FUNCTION_BLOCK Execute IMPLEMENTS ITF_PackMLState, ITF_States
VAR
	_MyContext : ITF_PackMLMachine;
	_MyNextState : ITF_PackMLState;
	_MyStoppingState : ITF_PackMLState;
	_MyAbortingState : ITF_PackMLState;
	_MyName : STRING(20) := 'Execute';
END_VAR

PROPERTY AbortingState : ITF_PackMLState
GET
AbortingState := _MyAbortingState;
END_GET
SET
_MyAbortingState := AbortingState;
END_SET
END_PROPERTY

METHOD CyclicLogic : BOOL
VAR_INPUT
END_VAR
END_METHOD

{warning 'add method implementation '}
METHOD EStop : BOOL
END_METHOD

{warning 'add property implementation'}
PROPERTY MyNextState : ITF_PackMLState
GET
MyNextState := _MyNextState;
END_GET
SET
_MyNextState := MyNextState;
END_SET
END_PROPERTY

PROPERTY MyStateName : String(20)
GET
MyStateName := _MyName;
END_GET
END_PROPERTY

{warning 'add method implementation '}
METHOD Reset : BOOL
END_METHOD

{warning 'add method implementation '}
METHOD SetContext : BOOL
VAR_INPUT
	context	: ITF_PackMLMachine;
END_VAR
_MyContext := context;
END_METHOD

{warning 'add method implementation '}
METHOD Start : BOOL
END_METHOD

{warning 'add method implementation '}
METHOD Stop : BOOL
END_METHOD

{warning 'add property implementation'}
PROPERTY StoppingState : ITF_PackMLState
GET
StoppingState := _MyStoppingState;
END_GET
SET
_MyStoppingState := StoppingState;
END_SET
END_PROPERTY

END_FUNCTION_BLOCK

(* stored: Version 1.1.0.1, ProductVersion 3.1.4024.12
   POU Execute: Id {16de238c-02d0-4654-b592-0c63039045d2}, SpecialFunc None
   Property AbortingState: Id {a5c15762-a08b-4161-91c2-5b5d8500ebc6}
   Get Get: Id {8849a4be-4f5c-408f-8893-220c57711478}
   Set Set: Id {d35cdb24-c26a-4df2-ac93-3d6a83189bfe}
   Method CyclicLogic: Id {ac050c99-a704-455e-9c5a-e556222f067a}
   Method EStop: Id {2ba6e0cd-1efe-4003-8123-65a9ba9b7ac2}
   Property MyNextState: Id {2d3d8db9-a44d-47ba-a9fd-8c0878cf2f5b}
   Get Get: Id {5d2e5776-26ac-4a8d-9a97-ef8b5054a217}
   Set Set: Id {b0111621-da13-46d4-85b1-9f62b318817a}
   Property MyStateName: Id {8976abae-eefc-4513-8348-4ffb6ed01903}
   Get Get: Id {0ffcb83e-153b-4248-94b8-c0ac0d69ac6e}
   Method Reset: Id {1a9cf0ec-8b14-4e8d-9539-992a9b7b2e78}
   Method SetContext: Id {1700c1be-96df-4ce8-8a27-f90db3bd76f2}
   Method Start: Id {42576e4a-c1d8-4012-9b36-1be3c4c250b5}
   Method Stop: Id {26dae254-0c3f-4d8e-8ed6-04c9be98f59b}
   Property StoppingState: Id {94f61d8a-f201-44ab-9c5d-1676d4b7878e}
   Get Get: Id {fcd83bcc-4566-4c4b-88c2-ce94446d7b5f}
   Set Set: Id {a8a29974-6336-4375-985e-b30003b343df} *)
